FUNCTION_BLOCK FB_NOTT_CO2_PRESSURE_CONTROL
VAR_INPUT
END_VAR
VAR_OUTPUT
END_VAR
VAR
	CO2_Valve:	FB_CRYO_VALVE_CTRL;
	
	// Pointers to valves
	ptrV:	 POINTER TO FB_CRYO_VALVE_CTRL;
	// Pointers to valve commands
	ptrVC:	 POINTER TO FB_CRYO_CMD_OVERRIDE;
	// Pointers to Enable flags for valves
	ptrEV:	 POINTER TO BOOL;
	
	cor_CO2_Valve:	FB_CRYO_CMD_OVERRIDE;
	bEnable_CO2_Valve:	BOOL := FALSE;
		
	
	
	stat:		T_NOTT_STAT;
	
	nCO2_Diff_Press_Sens AT %I*	:INT;
	lrCO2_Diff_Press_mbar:		LREAL;
	
	bConfigured:		BOOL := FALSE;
	
END_VAR



M_Configure();

M_ReadSensors();

M_Execute_Controller();

METHOD M_Configure : BOOL
VAR_INPUT
END_VAR


IF NOT bConfigured THEN




	ptrV := ADR(CO2_Valve);
	
	
	// Set pointers to Valve Commands - MUST!!!
	ptrVC	:= ADR(cor_CO2_Valve);
	
	ptrEV	:= ADR(bEnable_CO2_Valve);
	
	
	
	
	bConfigured := TRUE;


END_IF
END_METHOD

METHOD M_Execute_Controller : BOOL
VAR_INPUT
END_VAR
cor_CO2_Valve(in_bEnable := bEnable_CO2_Valve);	// Handling of PVV1 commands

CO2_Valve(
	in_sName			:= 'CO2_Valve', 
	in_bEnable			:= cor_CO2_Valve.out_bEnable,
	in_nFeedback		:= E_CRYO_BIN_ACT_FEEDBACK.ON_ONLY);
END_METHOD

METHOD M_ReadSensors : BOOL
VAR_INPUT
END_VAR


lrCO2_Diff_Press_mbar := nCO2_Diff_Press_Sens * 0.01;
END_METHOD

END_FUNCTION_BLOCK

(* stored: Version 1.1.0.1, ProductVersion 3.1.4024.14
   POU FB_NOTT_CO2_PRESSURE_CONTROL: Id {ed2768eb-fec2-4f1e-903e-ca4d99e4a92f}, SpecialFunc None
   Method M_Configure: Id {ac5d4578-9264-47ed-8c8d-ebcb3ba747ad}
   Method M_Execute_Controller: Id {6f90081b-56ca-47b4-b3a4-6fff259ba009}
   Method M_ReadSensors: Id {8803597c-1c5f-4621-9384-5ec6a2d9b9dc} *)
